{attribute 'qualified_only'}
VAR_GLOBAL
	
	robot:structRobot;

END_VAR

(* stored: Version 1.1.0.1, ProductVersion 3.1.4024.12
   GVL robotGlobals: Id {258cf7b6-e668-4946-9fc9-6d28e8d0ab60} *)
